// TIA Portal V19 export
FUNCTION "A0303_Spalla_Testa_CALL" : Void   // FC191, LAD
// stored: SetENOAutomatically false
   VAR CONSTANT
      MISSING : Int;
   END_VAR
BEGIN

REGION Network 1: Data In - Ax
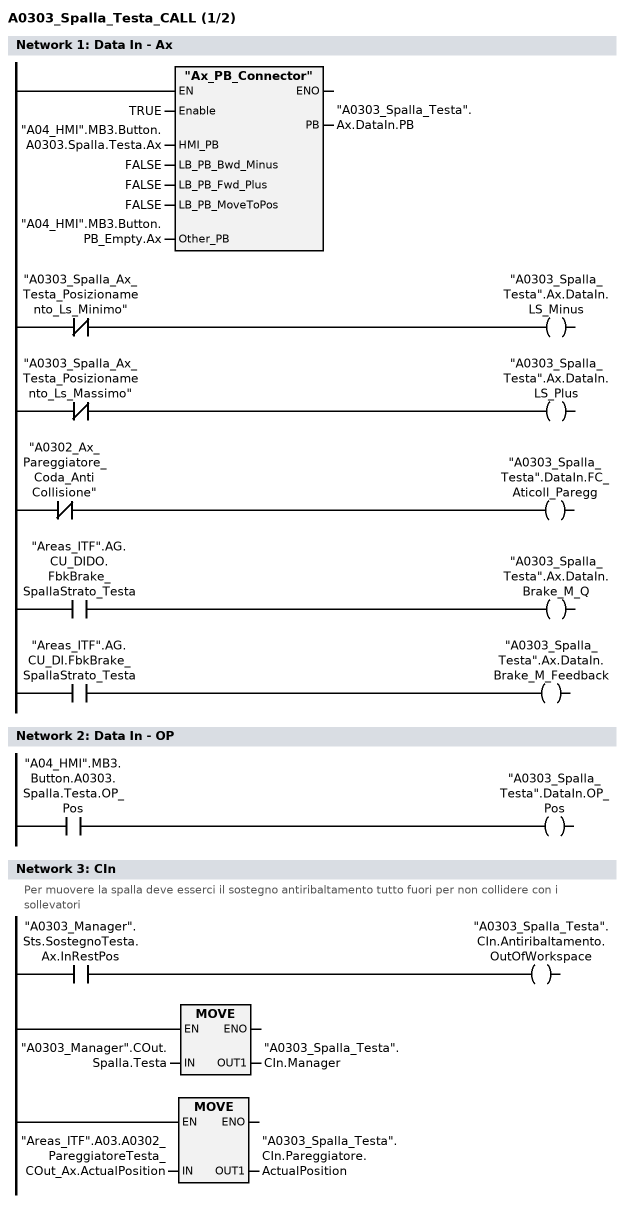
   RUNG wire#powerrail
      "Ax_PB_Connector"(Enable := TRUE, HMI_PB := "A04_HMI".MB3.Button.A0303.Spalla.Testa.Ax, LB_PB_Bwd_Minus := FALSE, LB_PB_Fwd_Plus := FALSE, LB_PB_MoveToPos := FALSE, Other_PB := "A04_HMI".MB3.Button.PB_Empty.Ax, PB => "A0303_Spalla_Testa".Ax.DataIn.PB)
   END_RUNG
   RUNG wire#powerrail
      I_Contact( "A0303_Spalla_Ax_Testa_Posizionamento_Ls_Minimo" )
      Coil( "A0303_Spalla_Testa".Ax.DataIn.LS_Minus )
   END_RUNG
   RUNG wire#powerrail
      I_Contact( "A0303_Spalla_Ax_Testa_Posizionamento_Ls_Massimo" )
      Coil( "A0303_Spalla_Testa".Ax.DataIn.LS_Plus )
   END_RUNG
   RUNG wire#powerrail
      I_Contact( "A0302_Ax_Pareggiatore_Coda_AntiCollisione" )
      Coil( "A0303_Spalla_Testa".DataIn.FC_Aticoll_Paregg )
   END_RUNG
   RUNG wire#powerrail
      Contact( "Areas_ITF".AG.CU_DIDO.FbkBrake_SpallaStrato_Testa )
      Coil( "A0303_Spalla_Testa".Ax.DataIn.Brake_M_Q )
   END_RUNG
   RUNG wire#powerrail
      Contact( "Areas_ITF".AG.CU_DI.FbkBrake_SpallaStrato_Testa )
      Coil( "A0303_Spalla_Testa".Ax.DataIn.Brake_M_Feedback )
   END_RUNG
   // the same network as SCL:
   "Ax_PB_Connector"(Enable := TRUE,
                     HMI_PB := "A04_HMI".MB3.Button.A0303.Spalla.Testa.Ax,
                     LB_PB_Bwd_Minus := FALSE,
                     LB_PB_Fwd_Plus := FALSE,
                     LB_PB_MoveToPos := FALSE,
                     Other_PB := "A04_HMI".MB3.Button.PB_Empty.Ax,
                     PB => "A0303_Spalla_Testa".Ax.DataIn.PB);
   "A0303_Spalla_Testa".Ax.DataIn.LS_Minus := NOT "A0303_Spalla_Ax_Testa_Posizionamento_Ls_Minimo";
   "A0303_Spalla_Testa".Ax.DataIn.LS_Plus := NOT "A0303_Spalla_Ax_Testa_Posizionamento_Ls_Massimo";
   "A0303_Spalla_Testa".DataIn.FC_Aticoll_Paregg := NOT "A0302_Ax_Pareggiatore_Coda_AntiCollisione";
   "A0303_Spalla_Testa".Ax.DataIn.Brake_M_Q := "Areas_ITF".AG.CU_DIDO.FbkBrake_SpallaStrato_Testa;
   "A0303_Spalla_Testa".Ax.DataIn.Brake_M_Feedback := "Areas_ITF".AG.CU_DI.FbkBrake_SpallaStrato_Testa;
END_REGION

REGION Network 2: Data In - OP
   RUNG wire#powerrail
      Contact( "A04_HMI".MB3.Button.A0303.Spalla.Testa.OP_Pos )
      Coil( "A0303_Spalla_Testa".DataIn.OP_Pos )
   END_RUNG
   // the same network as SCL:
   "A0303_Spalla_Testa".DataIn.OP_Pos := "A04_HMI".MB3.Button.A0303.Spalla.Testa.OP_Pos;
END_REGION

REGION Network 3: CIn
   // Per muovere la spalla deve esserci il sostegno antiribaltamento tutto fuori per non collidere con i sollevatori
   RUNG wire#powerrail
      Contact( "A0303_Manager".Sts.SostegnoTesta.Ax.InRestPos )
      Coil( "A0303_Spalla_Testa".CIn.Antiribaltamento.OutOfWorkspace )
   END_RUNG
   RUNG wire#powerrail
      Move(in := "A0303_Manager".COut.Spalla.Testa, out1 => "A0303_Spalla_Testa".CIn.Manager)
   END_RUNG
   RUNG wire#powerrail
      Move(in := "Areas_ITF".A03.A0302_PareggiatoreTesta_COut_Ax.ActualPosition, out1 => "A0303_Spalla_Testa".CIn.Pareggiatore.ActualPosition)
   END_RUNG
   // the same network as SCL:
   "A0303_Spalla_Testa".CIn.Antiribaltamento.OutOfWorkspace := "A0303_Manager".Sts.SostegnoTesta.Ax.InRestPos;
   "A0303_Spalla_Testa".CIn.Manager := "A0303_Manager".COut.Spalla.Testa;
   "A0303_Spalla_Testa".CIn.Pareggiatore.ActualPosition := "Areas_ITF".A03.A0302_PareggiatoreTesta_COut_Ax.ActualPosition;
END_REGION

REGION Network 4: HW
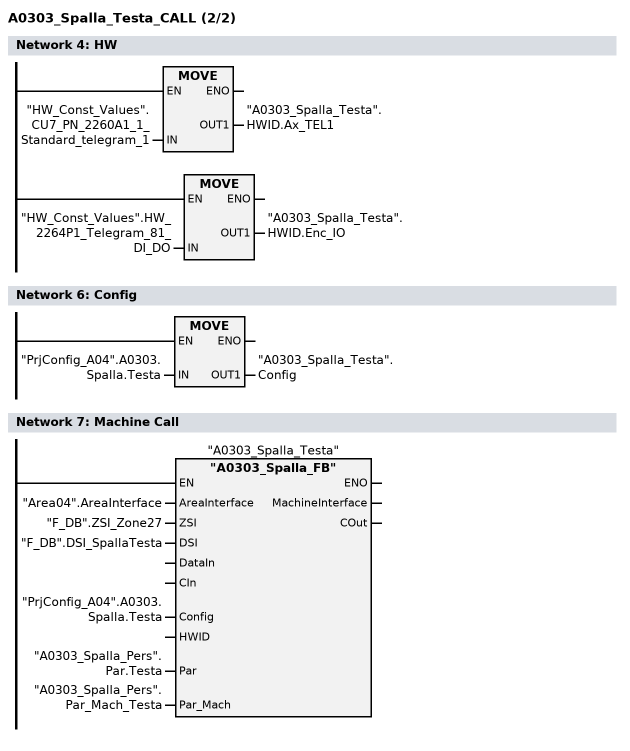
   RUNG wire#powerrail
      Move(in := "HW_Const_Values".CU7_PN_2260A1_1_Standard_telegram_1, out1 => "A0303_Spalla_Testa".HWID.Ax_TEL1)
   END_RUNG
   RUNG wire#powerrail
      Move(in := "HW_Const_Values".HW_2264P1_Telegram_81_DI_DO, out1 => "A0303_Spalla_Testa".HWID.Enc_IO)
   END_RUNG
   // the same network as SCL:
   "A0303_Spalla_Testa".HWID.Ax_TEL1 := "HW_Const_Values".CU7_PN_2260A1_1_Standard_telegram_1;
   "A0303_Spalla_Testa".HWID.Enc_IO := "HW_Const_Values".HW_2264P1_Telegram_81_DI_DO;
END_REGION

REGION Network 5 (SCL): Drive
   "A0303_Spalla_Testa".Ax.Drive.Infeed_ON := "Areas_ITF".AG.Infeed_Running;
   "A0303_Spalla_Testa".Ax.Drive.AccessPoint := "HW_Const_Values".CU7_PN_610A1_ModuleAccessPoint;
   "A0303_Spalla_Testa".Ax.Drive.AxisID := "CU7_ID_4_2260A1_1_2260M1";
   "A0303_Spalla_Testa".Ax.Drive.TokenChain := "TOKENCHAIN_CU7";
END_REGION

REGION Network 6: Config
   RUNG wire#powerrail
      Move(in := "PrjConfig_A04".A0303.Spalla.Testa, out1 => "A0303_Spalla_Testa".Config)
   END_RUNG
   // the same network as SCL:
   "A0303_Spalla_Testa".Config := "PrjConfig_A04".A0303.Spalla.Testa;
END_REGION

REGION Network 7: Machine Call
   RUNG wire#powerrail
      "A0303_Spalla_Testa"(AreaInterface := "Area04".AreaInterface, ZSI := "F_DB".ZSI_Zone27, DSI := "F_DB".DSI_SpallaTesta, DataIn :=, CIn :=, Config := "PrjConfig_A04".A0303.Spalla.Testa, HWID :=, Par := "A0303_Spalla_Pers".Par.Testa, Par_Mach := "A0303_Spalla_Pers".Par_Mach_Testa, MachineInterface =>, COut =>)
   END_RUNG
   // the same network as SCL:
   "A0303_Spalla_Testa"(AreaInterface := "Area04".AreaInterface,   // "A0303_Spalla_FB"
                        ZSI := "F_DB".ZSI_Zone27,
                        DSI := "F_DB".DSI_SpallaTesta,
                        Config := "PrjConfig_A04".A0303.Spalla.Testa,
                        Par := "A0303_Spalla_Pers".Par.Testa,
                        Par_Mach := "A0303_Spalla_Pers".Par_Mach_Testa);
END_REGION

REGION Network 8: >
END_REGION

REGION Network 9: >
END_REGION

REGION Network 10: >
END_REGION
END_FUNCTION
